// TwinCAT 3 PLC project Sample
// ProgramVersion: 3.1.4026.23
// libraries:
//   Tc2_Standard, * (Beckhoff Automation GmbH)
//   Tc2_System, * (Beckhoff Automation GmbH)
// project tree:
//   GVLs/ Device_1_Client_1.TcGVL
//   / PlcTask.TcTTO
//   POUs/ MAIN.TcPOU
//   POUs/OpcUaClient/ FB_Device_1_Client_1_Sample_Methods_MyObject_MyMethod.TcPOU
// real-time tasks:
//   TASK Device 1 (OPC UA Virtual)_Task_58: cycle T#40ms, priority 58, ADS port 350
//   TASK PlcTask: cycle T#10ms, priority 20, ADS port 351
// I/O:
//   DEVICE Device 1 (OPC UA Virtual), AmsNetId 192.168.179.145.2.1
// variable links:
//   Sample/Sample Instance <-> Device 1 (OPC UA Virtual)/Client #1
//     PlcTask Inputs/Device_1_Client_1.bConnected <-> Inputs/Status/Connected
//     PlcTask Inputs/Device_1_Client_1.bReadBusy <-> Inputs/Status/ReadBusy
//     PlcTask Inputs/Device_1_Client_1.nKeepAlives <-> Inputs/Status/KeepAlives
//     PlcTask Inputs/Device_1_Client_1.nStmState <-> Inputs/Status/StmState
//     PlcTask Outputs/Device_1_Client_1.bExecute <-> Outputs/Control/Execute
//     PlcTask Outputs/Device_1_Client_1.bResetStm <-> Outputs/Control/ResetStm
//     PlcTask Outputs/Device_1_Client_1.bWrite_Enable <-> Outputs/Control/Write Enable
//   Sample/Sample Instance <-> Device 1 (OPC UA Virtual)/Client #1/Sample.Arrays/MyArrayByteString
//     PlcTask Inputs/Device_1_Client_1.Sample_Arrays_MyArrayByteString <-> Inputs/Value
//     PlcTask Inputs/Device_1_Client_1.Sample_Arrays_errMyArrayByteString <-> Inputs/ErrorCode
//     PlcTask Inputs/Device_1_Client_1.Sample_Arrays_tsMyArrayByteString <-> Inputs/TimeStamp
//     PlcTask Outputs/Device_1_Client_1.Sample_Arrays_wMyArrayByteString <-> Outputs/Value
//   Sample/Sample Instance <-> Device 1 (OPC UA Virtual)/Client #1/Sample.Arrays/MyArrayInt32
//     PlcTask Inputs/Device_1_Client_1.Sample_Arrays_MyArrayInt32 <-> Inputs/Value
//     PlcTask Inputs/Device_1_Client_1.Sample_Arrays_errMyArrayInt32 <-> Inputs/ErrorCode
//     PlcTask Inputs/Device_1_Client_1.Sample_Arrays_tsMyArrayInt32 <-> Inputs/TimeStamp
//     PlcTask Outputs/Device_1_Client_1.Sample_Arrays_wMyArrayInt32 <-> Outputs/Value
//   Sample/Sample Instance <-> Device 1 (OPC UA Virtual)/Client #1/Sample.Methods.MyObject.MyMethod
//     PlcTask Inputs/Device_1_Client_1.Sample_Methods_MyObject_MyMethod.Output1 <-> Inputs/Output1
//     PlcTask Inputs/Device_1_Client_1.Sample_Methods_MyObject_MyMethod.Output2 <-> Inputs/Output2
//     PlcTask Inputs/Device_1_Client_1.Sample_Methods_MyObject_MyMethod.bBusy <-> Inputs/bBusy
//     PlcTask Inputs/Device_1_Client_1.Sample_Methods_MyObject_MyMethod.bDone <-> Inputs/bDone
//     PlcTask Inputs/Device_1_Client_1.Sample_Methods_MyObject_MyMethod.bError <-> Inputs/bError
//     PlcTask Inputs/Device_1_Client_1.Sample_Methods_MyObject_MyMethod.nErrorID <-> Inputs/nErrorID
//     PlcTask Outputs/Device_1_Client_1.Sample_Methods_MyObject_MyMethod.Input1 <-> Outputs/Input1
//     PlcTask Outputs/Device_1_Client_1.Sample_Methods_MyObject_MyMethod.Input2 <-> Outputs/Input2
//     PlcTask Outputs/Device_1_Client_1.Sample_Methods_MyObject_MyMethod.bExecute <-> Outputs/bExecute
//   Sample/Sample Instance <-> Device 1 (OPC UA Virtual)/Client #1/Sample.Scalars/MyInt16
//     PlcTask Inputs/Device_1_Client_1.Sample_Scalars_MyInt16 <-> Inputs/Value
//     PlcTask Inputs/Device_1_Client_1.Sample_Scalars_errMyInt16 <-> Inputs/ErrorCode
//     PlcTask Inputs/Device_1_Client_1.Sample_Scalars_tsMyInt16 <-> Inputs/TimeStamp
//     PlcTask Outputs/Device_1_Client_1.Sample_Scalars_wMyInt16 <-> Outputs/Value
//   Sample/Sample Instance <-> Device 1 (OPC UA Virtual)/Client #1/Sample.Scalars/MyInt32
//     PlcTask Inputs/Device_1_Client_1.Sample_Scalars_MyInt32 <-> Inputs/Value
//     PlcTask Inputs/Device_1_Client_1.Sample_Scalars_errMyInt32 <-> Inputs/ErrorCode
//     PlcTask Inputs/Device_1_Client_1.Sample_Scalars_tsMyInt32 <-> Inputs/TimeStamp
//     PlcTask Outputs/Device_1_Client_1.Sample_Scalars_wMyInt32 <-> Outputs/Value
//   Sample/Sample Instance <-> Device 1 (OPC UA Virtual)/Client #1/Sample.Scalars/MyInt32Static
//     PlcTask Inputs/Device_1_Client_1.Sample_Scalars_MyInt32Static <-> Inputs/Value
//     PlcTask Inputs/Device_1_Client_1.Sample_Scalars_errMyInt32Static <-> Inputs/ErrorCode
//     PlcTask Inputs/Device_1_Client_1.Sample_Scalars_tsMyInt32Static <-> Inputs/TimeStamp
//     PlcTask Outputs/Device_1_Client_1.Sample_Scalars_wMyInt32Static <-> Outputs/Value
//   Sample/Sample Instance <-> Device 1 (OPC UA Virtual)/Client #1/Sample.Scalars/MyInt64
//     PlcTask Inputs/Device_1_Client_1.Sample_Scalars_MyInt64 <-> Inputs/Value
//     PlcTask Inputs/Device_1_Client_1.Sample_Scalars_errMyInt64 <-> Inputs/ErrorCode
//     PlcTask Inputs/Device_1_Client_1.Sample_Scalars_tsMyInt64 <-> Inputs/TimeStamp
//     PlcTask Outputs/Device_1_Client_1.Sample_Scalars_wMyInt64 <-> Outputs/Value
//   Sample/Sample Instance <-> Device 1 (OPC UA Virtual)/Client #1/Sample.Scalars/MyString
//     PlcTask Inputs/Device_1_Client_1.Sample_Scalars_MyString <-> Inputs/Value
//     PlcTask Inputs/Device_1_Client_1.Sample_Scalars_errMyString <-> Inputs/ErrorCode
//     PlcTask Inputs/Device_1_Client_1.Sample_Scalars_tsMyString <-> Inputs/TimeStamp
//     PlcTask Outputs/Device_1_Client_1.Sample_Scalars_wMyString <-> Outputs/Value
//   Sample/Sample Instance <-> Device 1 (OPC UA Virtual)/Client #1/Sample.Structures/MyStructure
//     PlcTask Inputs/Device_1_Client_1.Sample_Structures_MyStructure <-> Inputs/Value
//     PlcTask Inputs/Device_1_Client_1.Sample_Structures_errMyStructure <-> Inputs/ErrorCode
//     PlcTask Inputs/Device_1_Client_1.Sample_Structures_tsMyStructure <-> Inputs/TimeStamp
//     PlcTask Outputs/Device_1_Client_1.Sample_Structures_wMyStructure <-> Outputs/Value

CONFIGURATION Sample
    RESOURCE PLC ON TwinCAT3
        TASK PlcTask(INTERVAL := T#10ms, PRIORITY := 20);
        PROGRAM MAIN WITH PlcTask : MAIN;
    END_RESOURCE
END_CONFIGURATION

// ---- GVLs/Device_1_Client_1.TcGVL
{attribute 'linkalways'}
VAR_GLOBAL
	{attribute 'TcLinkTo' := 'TIID^Device 1 (OPC UA Virtual)^Client #1^Inputs^Status^Connected'}
	bConnected AT %I* : BOOL;
	{attribute 'TcLinkTo' := 'TIID^Device 1 (OPC UA Virtual)^Client #1^Inputs^Status^ReadBusy'}
	bReadBusy AT %I* : BOOL;
	{attribute 'TcLinkTo' := 'TIID^Device 1 (OPC UA Virtual)^Client #1^Inputs^Status^KeepAlives'}
	nKeepAlives AT %I* : BYTE;
	{attribute 'TcLinkTo' := 'TIID^Device 1 (OPC UA Virtual)^Client #1^Inputs^Status^StmState'}
	nStmState AT %I* : BYTE;
	{attribute 'TcLinkTo' := 'TIID^Device 1 (OPC UA Virtual)^Client #1^Outputs^Control^ResetStm'}
	bResetStm AT %Q* : BOOL;
	{attribute 'TcLinkTo' := 'TIID^Device 1 (OPC UA Virtual)^Client #1^Outputs^Control^Execute'}
	bExecute AT %Q* : BOOL;
	{attribute 'TcLinkTo' := 'TIID^Device 1 (OPC UA Virtual)^Client #1^Outputs^Control^Write Enable'}
	bWrite_Enable AT %Q* : BOOL;


	{attribute 'TcLinkTo' := 'TIID^Device 1 (OPC UA Virtual)^Client #1^Sample.Arrays^MyArrayByteString^Inputs^Value'}
	Sample_Arrays_MyArrayByteString AT %I* : ARRAY [0..9] OF OpcUa_ByteString;
	{attribute 'TcLinkTo' := 'TIID^Device 1 (OPC UA Virtual)^Client #1^Sample.Arrays^MyArrayByteString^Inputs^TimeStamp'}
	Sample_Arrays_tsMyArrayByteString AT %I* : ULINT;
	{attribute 'TcLinkTo' := 'TIID^Device 1 (OPC UA Virtual)^Client #1^Sample.Arrays^MyArrayByteString^Inputs^ErrorCode'}
	Sample_Arrays_errMyArrayByteString AT %I* : UDINT;
	{attribute 'TcLinkTo' := 'TIID^Device 1 (OPC UA Virtual)^Client #1^Sample.Arrays^MyArrayByteString^Outputs^Value'}
	Sample_Arrays_wMyArrayByteString AT %Q* : ARRAY [0..9] OF OpcUa_ByteString;

	{attribute 'TcLinkTo' := 'TIID^Device 1 (OPC UA Virtual)^Client #1^Sample.Arrays^MyArrayInt32^Inputs^Value'}
	Sample_Arrays_MyArrayInt32 AT %I* : ARRAY [0..9] OF DINT;
	{attribute 'TcLinkTo' := 'TIID^Device 1 (OPC UA Virtual)^Client #1^Sample.Arrays^MyArrayInt32^Inputs^TimeStamp'}
	Sample_Arrays_tsMyArrayInt32 AT %I* : ULINT;
	{attribute 'TcLinkTo' := 'TIID^Device 1 (OPC UA Virtual)^Client #1^Sample.Arrays^MyArrayInt32^Inputs^ErrorCode'}
	Sample_Arrays_errMyArrayInt32 AT %I* : UDINT;
	{attribute 'TcLinkTo' := 'TIID^Device 1 (OPC UA Virtual)^Client #1^Sample.Arrays^MyArrayInt32^Outputs^Value'}
	Sample_Arrays_wMyArrayInt32 AT %Q* : ARRAY [0..9] OF DINT;


	{attribute 'TcLinkTo' := 'TIID^Device 1 (OPC UA Virtual)^Client #1^Sample.Structures^MyStructure^Inputs^Value'}
	Sample_Structures_MyStructure AT %I* : OpcUa_MyStructure;
	{attribute 'TcLinkTo' := 'TIID^Device 1 (OPC UA Virtual)^Client #1^Sample.Structures^MyStructure^Inputs^TimeStamp'}
	Sample_Structures_tsMyStructure AT %I* : ULINT;
	{attribute 'TcLinkTo' := 'TIID^Device 1 (OPC UA Virtual)^Client #1^Sample.Structures^MyStructure^Inputs^ErrorCode'}
	Sample_Structures_errMyStructure AT %I* : UDINT;
	{attribute 'TcLinkTo' := 'TIID^Device 1 (OPC UA Virtual)^Client #1^Sample.Structures^MyStructure^Outputs^Value'}
	Sample_Structures_wMyStructure AT %Q* : OpcUa_MyStructure;


	{attribute 'TcLinkTo' := 'TIID^Device 1 (OPC UA Virtual)^Client #1^Sample.Scalars^MyInt16^Inputs^Value'}
	Sample_Scalars_MyInt16 AT %I* : INT;
	{attribute 'TcLinkTo' := 'TIID^Device 1 (OPC UA Virtual)^Client #1^Sample.Scalars^MyInt16^Inputs^TimeStamp'}
	Sample_Scalars_tsMyInt16 AT %I* : ULINT;
	{attribute 'TcLinkTo' := 'TIID^Device 1 (OPC UA Virtual)^Client #1^Sample.Scalars^MyInt16^Inputs^ErrorCode'}
	Sample_Scalars_errMyInt16 AT %I* : UDINT;
	{attribute 'TcLinkTo' := 'TIID^Device 1 (OPC UA Virtual)^Client #1^Sample.Scalars^MyInt16^Outputs^Value'}
	Sample_Scalars_wMyInt16 AT %Q* : INT;

	{attribute 'TcLinkTo' := 'TIID^Device 1 (OPC UA Virtual)^Client #1^Sample.Scalars^MyInt32^Inputs^Value'}
	Sample_Scalars_MyInt32 AT %I* : DINT;
	{attribute 'TcLinkTo' := 'TIID^Device 1 (OPC UA Virtual)^Client #1^Sample.Scalars^MyInt32^Inputs^TimeStamp'}
	Sample_Scalars_tsMyInt32 AT %I* : ULINT;
	{attribute 'TcLinkTo' := 'TIID^Device 1 (OPC UA Virtual)^Client #1^Sample.Scalars^MyInt32^Inputs^ErrorCode'}
	Sample_Scalars_errMyInt32 AT %I* : UDINT;
	{attribute 'TcLinkTo' := 'TIID^Device 1 (OPC UA Virtual)^Client #1^Sample.Scalars^MyInt32^Outputs^Value'}
	Sample_Scalars_wMyInt32 AT %Q* : DINT;

	{attribute 'TcLinkTo' := 'TIID^Device 1 (OPC UA Virtual)^Client #1^Sample.Scalars^MyInt64^Inputs^Value'}
	Sample_Scalars_MyInt64 AT %I* : LINT;
	{attribute 'TcLinkTo' := 'TIID^Device 1 (OPC UA Virtual)^Client #1^Sample.Scalars^MyInt64^Inputs^TimeStamp'}
	Sample_Scalars_tsMyInt64 AT %I* : ULINT;
	{attribute 'TcLinkTo' := 'TIID^Device 1 (OPC UA Virtual)^Client #1^Sample.Scalars^MyInt64^Inputs^ErrorCode'}
	Sample_Scalars_errMyInt64 AT %I* : UDINT;
	{attribute 'TcLinkTo' := 'TIID^Device 1 (OPC UA Virtual)^Client #1^Sample.Scalars^MyInt64^Outputs^Value'}
	Sample_Scalars_wMyInt64 AT %Q* : LINT;

	{attribute 'TcLinkTo' := 'TIID^Device 1 (OPC UA Virtual)^Client #1^Sample.Scalars^MyString^Inputs^Value'}
	Sample_Scalars_MyString AT %I* : STRING(80);
	{attribute 'TcLinkTo' := 'TIID^Device 1 (OPC UA Virtual)^Client #1^Sample.Scalars^MyString^Inputs^TimeStamp'}
	Sample_Scalars_tsMyString AT %I* : ULINT;
	{attribute 'TcLinkTo' := 'TIID^Device 1 (OPC UA Virtual)^Client #1^Sample.Scalars^MyString^Inputs^ErrorCode'}
	Sample_Scalars_errMyString AT %I* : UDINT;
	{attribute 'TcLinkTo' := 'TIID^Device 1 (OPC UA Virtual)^Client #1^Sample.Scalars^MyString^Outputs^Value'}
	Sample_Scalars_wMyString AT %Q* : STRING(80);

	{attribute 'TcLinkTo' := 'TIID^Device 1 (OPC UA Virtual)^Client #1^Sample.Scalars^MyInt32Static^Inputs^Value'}
	Sample_Scalars_MyInt32Static AT %I* : DINT;
	{attribute 'TcLinkTo' := 'TIID^Device 1 (OPC UA Virtual)^Client #1^Sample.Scalars^MyInt32Static^Inputs^TimeStamp'}
	Sample_Scalars_tsMyInt32Static AT %I* : ULINT;
	{attribute 'TcLinkTo' := 'TIID^Device 1 (OPC UA Virtual)^Client #1^Sample.Scalars^MyInt32Static^Inputs^ErrorCode'}
	Sample_Scalars_errMyInt32Static AT %I* : UDINT;
	{attribute 'TcLinkTo' := 'TIID^Device 1 (OPC UA Virtual)^Client #1^Sample.Scalars^MyInt32Static^Outputs^Value'}
	Sample_Scalars_wMyInt32Static AT %Q* : DINT;

	{attribute 'TcLinkTo' := '.nErrorID:=TIID^Device 1 (OPC UA Virtual)^Client #1^Sample.Methods.MyObject.MyMethod^Inputs^nErrorID;
	                          .bDone:=TIID^Device 1 (OPC UA Virtual)^Client #1^Sample.Methods.MyObject.MyMethod^Inputs^bDone;
	                          .bBusy:=TIID^Device 1 (OPC UA Virtual)^Client #1^Sample.Methods.MyObject.MyMethod^Inputs^bBusy;
	                          .bError:=TIID^Device 1 (OPC UA Virtual)^Client #1^Sample.Methods.MyObject.MyMethod^Inputs^bError;
	                          .Output1:=TIID^Device 1 (OPC UA Virtual)^Client #1^Sample.Methods.MyObject.MyMethod^Inputs^Output1;
	                          .Output2:=TIID^Device 1 (OPC UA Virtual)^Client #1^Sample.Methods.MyObject.MyMethod^Inputs^Output2;
	                          .bExecute:=TIID^Device 1 (OPC UA Virtual)^Client #1^Sample.Methods.MyObject.MyMethod^Outputs^bExecute;
	                          .Input1:=TIID^Device 1 (OPC UA Virtual)^Client #1^Sample.Methods.MyObject.MyMethod^Outputs^Input1;
	                          .Input2:=TIID^Device 1 (OPC UA Virtual)^Client #1^Sample.Methods.MyObject.MyMethod^Outputs^Input2'}
	Sample_Methods_MyObject_MyMethod : FB_Device_1_Client_1_Sample_Methods_MyObject_MyMethod;

END_VAR

// ---- POUs/MAIN.TcPOU
PROGRAM MAIN
VAR
	(* Variable declarations used for method call sample *)
	bCallMethod : BOOL;
	Input1 : INT := 21;
	Input2 : DINT := 21;
	Output1 : INT;
	Output2 : DINT;
	nMethodCallState : UINT;
	
	(* Variable declarations used for write sample *)
	bToggleWrite : BOOL;
END_VAR

CASE nMethodCallState OF

    0: // Init, waiting for bCallMethod to be set to TRUE
        IF bCallMethod THEN
            bCallMethod := FALSE;
            nMethodCallState := nMethodCallState + 1;
        END_IF

    1: // Calling the method
        Sample_Methods_MyObject_MyMethod(
            bExecute := TRUE,
            Input1 := Input1,
            Input2 := Input2
        );
		// Note that the OPC UA Client driver usually runs slower than the PLC task. 
		// This can be configured on the task that is linked with the OPC UA Client device. (In this example: Device 1 (OPC UA Virtual)_Task_58)
		// Therefore, it may take several PLC cycles until the driver detects the rising edge on bExecute and starts processing the method call. 
		// Wait until bBusy becomes TRUE before continuing, because this confirms that the method call has actually been accepted/started by the driver.
		IF Sample_Methods_MyObject_MyMethod.bBusy THEN
			nMethodCallState := nMethodCallState + 1;	
		END_IF

    2: // Waiting for method execution to complete
        Sample_Methods_MyObject_MyMethod(
            bExecute := TRUE,
            Output1 => Output1,
            Output2 => Output2
        );
        IF NOT Sample_Methods_MyObject_MyMethod.bBusy THEN
            IF NOT Sample_Methods_MyObject_MyMethod.bError THEN
				Sample_Methods_MyObject_MyMethod(bExecute := FALSE);
                nMethodCallState := 0;
            ELSE
                nMethodCallState := 255;
            END_IF
        END_IF

    255: // Error state

END_CASE

// Toggle cyclic write commands - cycle time is configured via a corresponding setting on the virtual OPC UA client device
IF bToggleWrite THEN
	bToggleWrite := FALSE;
	Device_1_Client_1.bWrite_Enable := NOT Device_1_Client_1.bWrite_Enable; // Activate write commands on virtual OPC UA client device
END_IF
Device_1_Client_1.Sample_Scalars_wMyInt32Static := Device_1_Client_1.Sample_Scalars_wMyInt32Static + 1; // Set new value for variable

END_PROGRAM

// ---- POUs/OpcUaClient/FB_Device_1_Client_1_Sample_Methods_MyObject_MyMethod.TcPOU
FUNCTION_BLOCK  FB_Device_1_Client_1_Sample_Methods_MyObject_MyMethod
VAR_INPUT
	bExecute AT %Q* : BOOL;
	Input1 AT %Q* : INT;
	Input2 AT %Q* : DINT;
END_VAR
VAR_OUTPUT
	nErrorID AT %I* : DINT;
	bDone AT %I* : BOOL;
	bBusy AT %I* : BOOL;
	bError AT %I* : BOOL;
	Output1 AT %I* : INT;
	Output2 AT %I* : DINT;
END_VAR

END_FUNCTION_BLOCK
